VAR_GLOBAL
	fbMachineLogger : FB_FileLogger;
	fbMachineTime	: AliasOnlyThisProject;
END_VAR

(* stored: Version 1.1.0.1, ProductVersion 3.1.4024.12
   GVL GVL: Id {9bbaf649-16ad-4638-9817-6a7ae1f93f6d} *)
